// TwinCAT 3 PLC project Plc
// Company: TcOpenGroup
// Author: TcOpenGroup
// ProjectVersion: 0.0.0.1
// ProgramVersion: 3.1.4024.12
// libraries:
//   Tc2_Standard, * (Beckhoff Automation GmbH)
//   Tc2_System, * (Beckhoff Automation GmbH)
//   Tc3_Module, * (Beckhoff Automation GmbH)
//   TcoCore, 0.4.0.229 (Vortex.Library)
//   TcoPneumatics, 0.4.0.229 (Vortex.Library)
// project tree:
//   Components/ fbPiston.TcPOU, fbPistonMoveTask.TcPOU, IPistonHorizontal.TcIO (not stored), IPistonVertical.TcIO (not stored), IPistonGripper.TcIO (not stored)
//   / PlcTask.TcTTO
//   POUs/ MAIN.TcPOU, Station001.TcPOU, Station001_Components.TcPOU (not stored), Station001_Sequencer.TcPOU
// real-time tasks:
//   TASK PlcTask: cycle T#10ms, priority 20, ADS port 350

CONFIGURATION Plc
    RESOURCE PLC ON TwinCAT3
        TASK PlcTask(INTERVAL := T#10ms, PRIORITY := 20);
        PROGRAM MAIN WITH PlcTask : MAIN;
    END_RESOURCE
END_CONFIGURATION

// ---- POUs/MAIN.TcPOU
PROGRAM MAIN
VAR
	_station001 : Station001;
END_VAR

_station001.Run();

END_PROGRAM

// ---- POUs/Station001.TcPOU
FUNCTION_BLOCK Station001 EXTENDS TcoCore.TcoContext
VAR
	_components : Station001_Components(THIS^);
	_sequence : Station001_Sequencer(THIS^, FALSE, _components);
END_VAR

(*~
	<docu>
		<summary>
			Main method of the TcoContext. This is the entry point of any control logic that belongs to this context. 
			The call of this method is ensured by calling the <c>InstanceName.Run()</c> method, and it must not be called explicitly.
			This method is abstract, and it must be overridden in derived block.
		</summary>
	</docu>
~*)
METHOD PROTECTED  Main
_sequence.Run();
END_METHOD

END_FUNCTION_BLOCK

// ---- POUs/Station001_Sequencer.TcPOU
FUNCTION_BLOCK Station001_Sequencer EXTENDS TcoCore.TcoSequencer
VAR
	components : REFERENCE TO Station001_Components;
END_VAR

VAR
	_switchToStep : BOOL;
	_failedToLoad : BOOL;
END_VAR

METHOD FB_init : BOOL
VAR_INPUT
	bInitRetains : BOOL; // if TRUE, the retain variables are initialized (warm start / cold start)
	bInCopyCode : BOOL;  // if TRUE, the instance afterwards gets moved into the copy code (online change)
	Parent : ITcoObject;
	DoEnableAutoRestore : BOOL; 
	refComponents : REFERENCE TO Station001_Components;
END_VAR
Components REF= refComponents;
END_METHOD

METHOD Init
VAR_INPUT
END_VAR
components();

IF(_switchToStep) THEN
	THIS^._stepModeControler.ChangeState(TcoCore.eSequencerMode.StepMode);
	THIS^.Messenger.Notify('Sequencer is in step mode');
ELSE
	THIS^._stepModeControler.ChangeState(TcoCore.eSequencerMode.CyclicMode);
END_IF




IF(Step(0, 
		TRUE, 
		'INIT')) THEN
//-----------------------------------------------------
	THIS^.StepCompleteWhen(TRUE);
//-----------------------------------------------------	
END_IF
END_METHOD

(*~
	<docu>
		<summary>
			Main method of the sequener. Custom code needs to be placed here. The sequencer is executed by call of InstanceName.Run() method.
			This method is abstract, and it must be overridden in derived block.
		</summary>
	</docu>
~*)
METHOD  Main : BOOL
Init();

IF(Step(100, 
		TRUE, 
		'MOVE ALL CYLINDERS TO GROUND POSITION')) THEN
//-----------------------------------------------------
	StepCompleteWhen(components.Vertical.MoveUp().Done AND_THEN 
					 components.Horizontal.MoveLeft().Done AND_THEN 
					 components.Gripper.Open().Done);
//-----------------------------------------------------	
END_IF


IF(Step(200, 
		TRUE, 
		'MOVE VERTICAL CYLINDER DOWN')) THEN
//-----------------------------------------------------
	StepCompleteWhen(components.Vertical.MoveDown().Done);
//-----------------------------------------------------	
END_IF


IF(Step(300, 
		TRUE, 
		'CLOSE GRIPPER')) THEN
//-----------------------------------------------------
	IF(components.Gripper.Close().Done) THEN
		IF(_failedToLoad) THEN
			RequestStep(100);
		ELSE
			StepCompleteWhen(TRUE);	
		END_IF;	
		
	END_IF;		
//-----------------------------------------------------	
END_IF

IF(Step(400, 
		TRUE, 
		'MOVE VERTICAL CYLINDER UP')) THEN
//-----------------------------------------------------
	StepCompleteWhen(components.Vertical.MoveUp().Done);
//-----------------------------------------------------	
END_IF

IF(Step(500, 
		TRUE, 
		'MOVE HORIZONTAL CYLINDER TO UNLOAD POSITION')) THEN
//-----------------------------------------------------
	StepCompleteWhen(components.Horizontal.MoveRight().Done);
//-----------------------------------------------------	
END_IF

IF(Step(600, 
		TRUE, 
		'MOVE VERTICAL CYLINDER DOWN')) THEN
//-----------------------------------------------------
	StepCompleteWhen(components.Vertical.MoveDown().Done);
//-----------------------------------------------------	
END_IF

IF(Step(700, 
		TRUE, 
		'OPEN GRIPPER')) THEN
//-----------------------------------------------------
	StepCompleteWhen(components.Gripper.Open().Done);
//-----------------------------------------------------	
END_IF

IF(Step(800, 
		TRUE, 
		'CLOSE SEQUENCE')) THEN
//-----------------------------------------------------
	SequenceComplete();
//-----------------------------------------------------	
END_IF
END_METHOD

METHOD OnStateChange
VAR_INPUT
	PreviousState	: INT;
	NewState 		: INT;
END_VAR
// THIS^.Restore();
_stepModeControler._stepForward.Restore();
_stepModeControler._stepBackward.Restore();

IF(_stepModeControler._stepIn.Done) THEN _stepModeControler._stepIn.Restore(); END_IF;

components._simTimer(IN := FALSE);
END_METHOD

END_FUNCTION_BLOCK

// ---- Components/fbPiston.TcPOU
FUNCTION_BLOCK fbPiston EXTENDS TcoCore.TcoComponent
VAR_INPUT
	iHomePositionSensor : BOOL;
	iWorkPositionSensor : BOOL;	
END_VAR

VAR_OUTPUT
	qHomePositionActuator : BOOL;
	qWorkPositionActuator : BOOL;		
END_VAR

VAR
	_moveHomeTask : fbPistonMoveTask(THIS^);
	_moveWorkTask : fbPistonMoveTask(THIS^);
END_VAR

_moveHomeTask(PositionSensor := iHomePositionSensor, MoveToPositionSignal := qHomePositionActuator, InverseSignal := qWorkPositionActuator);
_moveWorkTask(PositionSensor := iWorkPositionSensor, MoveToPositionSignal := qWorkPositionActuator, InverseSignal := qHomePositionActuator);

METHOD Close : TcoCore.ITcoTask
Close := MoveToHome();
END_METHOD

METHOD PROTECTED Manual
VAR_INPUT
END_VAR
END_METHOD

METHOD MoveLeft : TcoCore.ITcoTask
MoveLeft := MoveToWork();
END_METHOD

METHOD MoveRight : TcoCore.ITcoTask
MoveRight := MoveToHome();
END_METHOD

METHOD PROTECTED MoveToHome : TcoCore.ITcoTask
MoveToHome := THIS^._moveHomeTask.Invoke();
END_METHOD

METHOD PROTECTED MoveToWork : TcoCore.ITcoTask
MoveToWork := THIS^._moveWorkTask.Invoke();
END_METHOD

METHOD Open : TcoCore.ITcoTask
Open := MoveToWork();
END_METHOD

METHOD  Restore : ITcoRestorable
THIS^._moveHomeTask.Restore();
THIS^._moveWorkTask.Restore();
END_METHOD

END_FUNCTION_BLOCK

// ---- Components/fbPistonMoveTask.TcPOU
FUNCTION_BLOCK fbPistonMoveTask EXTENDS TcoCore.TcoTask
VAR_INPUT
	PositionSensor : BOOL;
END_VAR
VAR_IN_OUT
	MoveToPositionSignal : BOOL;
	InverseSignal : BOOL;	
END_VAR

IF(THIS^.Execute())THEN
	THIS^.Messenger.Debug('Cylinder is moving, extremity sensor not reached yet.');
	InverseSignal := FALSE;
	MoveToPositionSignal := TRUE;
	THIS^.DoneWhen(PositionSensor);
END_IF

END_FUNCTION_BLOCK
